FUNCTION_BLOCK T_CartesianRobotProductionMode EXTENDS T_NamedBase IMPLEMENTS I_PackMode
VAR
	_cartesianRobot : I_CartesianRobotModule;
END_VAR

METHOD Initialise
VAR_INPUT
	CartesianRobotModule : I_CartesianRobotModule; 
END_VAR
_cartesianRobot := CartesianRobotModule;
END_METHOD

END_FUNCTION_BLOCK

(* stored: Version 1.1.0.1, ProductVersion 3.1.4024.12
   POU T_CartesianRobotProductionMode: Id {fc0ef1d1-1bdb-4894-b875-0df0fa4cabdc}, SpecialFunc None
   Method Initialise: Id {ad5d7965-df9b-482a-9a84-634752d60994} *)
